(* IEC 61131-3 sources: CodesysTest/alpha/export/Pro18_1174_Win10.dev/Plc Logic/Application/Motors/Applied Motion/FB_AppliedMotionStepServoTCP.pou, 1 file *)

(* ---- MoveToPosition.m.st ---- *)
(*#-#-#-#-#-#-#-#-#-#---Declaration---#-#-#-#-#-#-#-#-#-#-#-#-#*)

METHOD MoveToPosition
VAR_INPUT
    (*Position to move to in inches*)
    position    : REAL;
    (*Acceleration in RPM/sec*)
    acceleration    : INT;
    (*Deceleration in RPM/sec*)
    deceleration    : INT;
    (*Velocity in .25RPM*)
    velocity    : INT;
END_VAR
(*#-#-#-#-#-#-#-#-#-#---Implementation---#-#-#-#-#-#-#-#-#-#-#-#-#*)

//This method preps the data to send to the drive and triggers the send.
//Set distance and unpack to prep data to send to motor
distanceToMoveInSteps.rawValue := REAL_TO_DINT((position) * stepsPerInchSetpoint);
IF reversePolarity THEN
    distanceToMoveInSteps.rawValue := distanceToMoveInSteps.rawValue * -1;
END_IF
commandSuccessful := FALSE;
ModbusLongHandler.Unpack(distanceToMoveInSteps);
sendMoveCommand.acceleration := acceleration;
sendMoveCommand.deceleration := deceleration;
sendMoveCommand.velocity := velocity;
sendMoveCommand.distanceHighWord := distanceToMoveInSteps.highWord;
sendMoveCommand.distanceLowWord := distanceToMoveInSteps.lowWord;
sendMoveCommand.opcode := STEP_SERVO_OPCODES.FEED_TO_POSITION;
sendMoveCommand.Execute();
